TYPE (* REAL Value+Status *)
  (* Standard: 61499 Demo ITA; ApplicationDomain: Process Control; Type: Data Type *)
  (* Version 0.1, 2000-05-16, JHC, Rockwell Automation, File type changed to ".dtp" *)
  (* Version 0.0, 2000-04-12, JHC, Rockwell Automation *)
  (* Compiler header: package fb.rt.ita; *)
  (* Compiler Java IBM VisualAge 3.0 *)
  (* ASN.1 tag PRIVATE 10 *)
  REAL_VS : STRUCT
    VALUE : REAL;
    STATUS : BYTE;
  END_STRUCT;
END_TYPE
